FUNCTION_BLOCK LinearVelocity EXTENDS SM_LinearVelocity
VAR_INPUT
END_VAR
VAR_OUTPUT
END_VAR
VAR
    testVar : INT;
END_VAR

SUPER^();

END_FUNCTION_BLOCK

(* stored: Version 1.1.0.1, ProductVersion 3.1.4018.2
   POU LinearVelocity: Id {333d75b2-8370-4400-9313-e40e808ba083}, SpecialFunc None *)
